(* Schneider Machine Expert - Basic project test2, file version 1.9.0.0 *)
(* ProjectInformations: Name=New project *)

HARDWARE
  Cpu 0: TM221CE16R
  EthernetConfiguration: NetworkName=M221, IpAllocationMode=FixedAddress, IpAddress=0.0.0.0, SubnetMask=0.0.0.0
  SerialLineConfiguration: Baud=Baud19200, Parity=ParityEven, DataBits=DataBits8, StopBits=StopBits1, PhysicalMedium=PhysicalMediumRs485, TransmissionMode=TransmissionModeModbusRtu, SlaveId=1, Addressing=SlaveAddressing
  MastTask: UsePeriodScanMode=false, PeriodScan=100
  FastTask: Period=255
  CpuBehavior: StartingMode=StartAsPreviousState, AutoSaveRamOnEeprom=true, WatchdogPeriod=250

SYMBOLS  (address, symbol, comment, settings)

POU New POU
  (* SectionNumber=1 *)

// Rung 0
  LD %I0.0
  ST %Q0.0
  // as ST:
  //   %Q0.0 := %I0.0;

// Rung 1
  LD %Q0.0
  ST %M0
  // as ST:
  //   %M0 := %Q0.0;

// Rung 2
  LD %I0.1
  S %M1
  // as ST:
  //   IF %I0.1 THEN %M1 := TRUE; END_IF;

// Rung 3
  LD %I0.2
  R %M1
  // as ST:
  //   IF %I0.2 THEN %M1 := FALSE; END_IF;
